// TIA Portal V19 export
TYPE "SpeedMotor_Ctrl"
// stored: Access Published
   STRUCT
      SafeStop : Bool;   // Emergency stop (device in safe state)
      Rst : Bool;   // Reset alarms
      Power : Bool;   // Power axis command
      MovePlus : Bool;   // Move plus direction command
      MoveMinus : Bool;   // Move minus direction command
      Velocity : LReal;   // Velolcity (rpm)
      Acceleration : LReal;   // Acceleration (rpm/s2)
      Deceleration : LReal;   // Deceleration (rpm/s2)
   END_STRUCT;
END_TYPE
